(* IEC 61131-3 sources: Daniele1996.github.io/AUTOMATION_AND_SOFTWARE_DESIGN_PATTERN/AUTOMATION_STUDIO/Task2/Logical/Conveyor, 3 files *)

(* ---- Types.typ ---- *)
TYPE
	Conveyor_States: (
		Conveyor_ready_to_be_initialized,
		Conveyor_initializing,
		Conveyor_ready_to_be_enabled,
		Conveyor_enabling,
		Conveyor_ready_to_be_disabled,
		Conveyor_on_phase_stopping
	);
END_TYPE

(* ---- Main.st ---- *)
PROGRAM _INIT
	(* Insert code here *)

END_PROGRAM

PROGRAM _CYCLIC
	(* Insert code here *)
	CASE state OF
		Conveyor_ready_to_be_initialized:
			IF Conveyor_Handler.Initialize THEN
				Axis_Enable := TRUE;

				state := Conveyor_initializing;
			END_IF;

		Conveyor_initializing:
			IF NOT Axis_Enable THEN
				Conveyor_Handler.Initialize := FALSE;

				state := Conveyor_ready_to_be_enabled;
			END_IF;

		Conveyor_ready_to_be_enabled:
			IF Conveyor_Handler.Enable THEN
				Axis_Command := AXIS_MOVE_VELOCITY;

				state := Conveyor_enabling;
			END_IF;

		Conveyor_enabling:
			IF Axis_Command_Executed THEN
				Conveyor_Handler.Enable := FALSE;

				state := Conveyor_ready_to_be_disabled;
			END_IF;

		Conveyor_ready_to_be_disabled:
			IF Conveyor_Handler.On_Phase_Stop THEN
				Axis_Command := AXIS_STOP;

				state := Conveyor_on_phase_stopping;
			END_IF;

		Conveyor_on_phase_stopping:
			IF NOT Conveyor_Handler.On_Phase_Stop THEN

				state := Conveyor_ready_to_be_enabled;
			END_IF;
	END_CASE;

	Conveyor.Slave	:= ADR(gConveyor);

	Conveyor.AxisEnable_in := Axis_Enable;
	Conveyor.AxisCommand := Axis_Command;

	Conveyor.Velocity	:= CONVEYOR_VELOCITY;
	Conveyor.Acceleration	:= CONVEYOR_ACCELLERATION;
	Conveyor.Deceleration	:= CONVEYOR_DEACCELLERATION;

	Conveyor();

	Axis_Enable := Conveyor.AxisEnable_out;
	Axis_Command_Executed := Conveyor.CommandExecuted;
	CONVEYOR_POSITION := Conveyor.ActualPosition;
	CONVEYOR_ACTUAL_VELOCITY := REAL_TO_INT(Conveyor.ActualVelocity);

	ComTCP_SimOutputs.Shaft_0_ACT_POS := CONVEYOR_POSITION;

END_PROGRAM

PROGRAM _EXIT
	(* Insert code here *)

END_PROGRAM

(* ---- Variables.var ---- *)
VAR
	Conveyor : gAxis;
END_VAR

VAR
	state: Conveyor_States := Conveyor_ready_to_be_initialized;
END_VAR

VAR
	Axis_Command : WORD := AXIS_NULL_COMMAND;
	Axis_Command_Executed : BOOL;
	Axis_Enable : BOOL;
END_VAR

VAR
	CONVEYOR_POSITION : REAL;
	CONVEYOR_ACTUAL_VELOCITY : INT;
	CONVEYOR_ACCELLERATION : REAL := 100;
	CONVEYOR_DEACCELLERATION : REAL := 100;
	CONVEYOR_DISTANCE : REAL := 100;
END_VAR

VAR CONSTANT
	AXIS_NULL_COMMAND : WORD := 0;
	AXIS_MOVE_VELOCITY : WORD := 1;
	AXIS_MOVE_ADDITIVE : WORD := 2;
	AXIS_CAM_IN : WORD := 3;
	AXIS_STOP : WORD := 4;
END_VAR
